FUNCTION_BLOCK SludgeBufferBasic (* Basic Function Block Type *)
  (* Standard: 61499-2 *)
  (* Version 0.0, 6/29/2026, Schneider Electric, Template *)
  PACKAGE SE.Nereda;
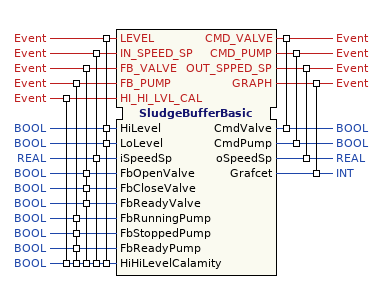
  EVENT_INPUT
    LEVEL WITH HiLevel, LoLevel, HiHiLevelCalamity;
    IN_SPEED_SP WITH iSpeedSp, HiHiLevelCalamity;
    FB_VALVE WITH FbOpenValve, FbCloseValve, FbReadyValve, HiHiLevelCalamity;
    FB_PUMP WITH FbRunningPump, FbStoppedPump, FbReadyPump, HiHiLevelCalamity;
    HI_HI_LVL_CAL WITH HiHiLevelCalamity;
  END_EVENT
  EVENT_OUTPUT
    CMD_VALVE WITH CmdValve;
    CMD_PUMP WITH CmdPump;
    OUT_SPPED_SP WITH oSpeedSp;
    GRAPH WITH Grafcet;
  END_EVENT
  VAR_INPUT
    HiLevel : BOOL;
    LoLevel : BOOL;
    iSpeedSp : REAL;
    FbOpenValve : BOOL;
    FbCloseValve : BOOL;
    FbReadyValve : BOOL;
    FbRunningPump : BOOL;
    FbStoppedPump : BOOL;
    FbReadyPump : BOOL;
    HiHiLevelCalamity : BOOL;
  END_VAR
  VAR_OUTPUT
    CmdValve : BOOL;
    CmdPump : BOOL;
    oSpeedSp : REAL;
    Grafcet : INT;
  END_VAR
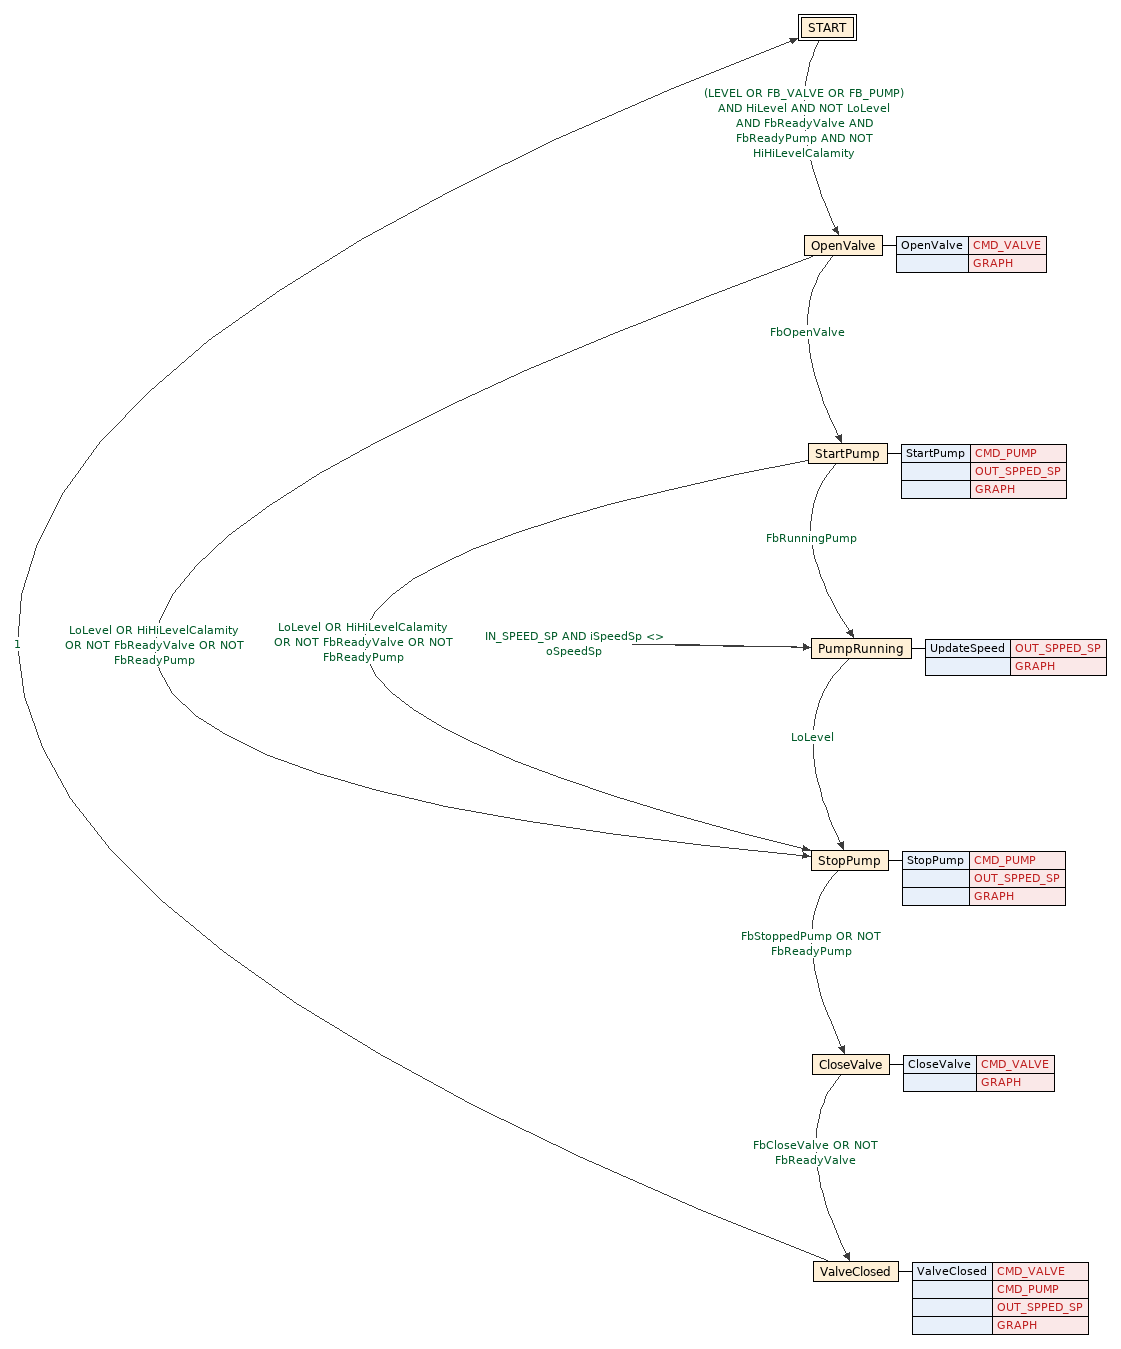
  EC_STATES
    START; (* Initial State *)
    OpenValve : OpenValve -> CMD_VALVE, -> GRAPH;
    StartPump : StartPump -> CMD_PUMP, -> OUT_SPPED_SP, -> GRAPH;
    PumpRunning : UpdateSpeed -> OUT_SPPED_SP, -> GRAPH;
    StopPump : StopPump -> CMD_PUMP, -> OUT_SPPED_SP, -> GRAPH;
    CloseValve : CloseValve -> CMD_VALVE, -> GRAPH;
    ValveClosed : ValveClosed -> CMD_VALVE, -> CMD_PUMP, -> OUT_SPPED_SP, -> GRAPH;
  END_STATES
  EC_TRANSITIONS
    START TO OpenValve := (LEVEL OR FB_VALVE OR FB_PUMP) AND HiLevel AND NOT LoLevel AND FbReadyValve AND FbReadyPump AND NOT HiHiLevelCalamity;
    OpenValve TO StartPump := FbOpenValve;
    StartPump TO PumpRunning := FbRunningPump;
    PumpRunning TO PumpRunning := IN_SPEED_SP AND iSpeedSp <> oSpeedSp;
    PumpRunning TO StopPump := LoLevel;
    StopPump TO CloseValve := FbStoppedPump OR NOT FbReadyPump;
    CloseValve TO ValveClosed := FbCloseValve OR NOT FbReadyValve;
    ValveClosed TO START := 1;
    StartPump TO StopPump := LoLevel OR HiHiLevelCalamity OR NOT FbReadyValve OR NOT FbReadyPump;
    OpenValve TO StopPump := LoLevel OR HiHiLevelCalamity OR NOT FbReadyValve OR NOT FbReadyPump;
  END_TRANSITIONS
  ALGORITHM OpenValve IN ST:
;
CmdValve := TRUE;
Grafcet := 1;
  END_ALGORITHM
  ALGORITHM StartPump IN ST:
;
CmdPump := TRUE;
oSpeedSp := iSpeedSp;
Grafcet := 2;
  END_ALGORITHM
  ALGORITHM UpdateSpeed IN ST:
;
oSpeedSp := iSpeedSp;
Grafcet := 3;
  END_ALGORITHM
  ALGORITHM StopPump IN ST:
;
CmdPump := FALSE;
oSpeedSp := 0;
Grafcet := 4;
  END_ALGORITHM
  ALGORITHM CloseValve IN ST:
;
CmdValve := FALSE;
Grafcet := 5;
  END_ALGORITHM
  ALGORITHM ValveClosed IN ST:
;
CmdValve := FALSE;
CmdPump := FALSE;
oSpeedSp := 0;
Grafcet := 6;
  END_ALGORITHM
END_FUNCTION_BLOCK
